TYPE M2MultiplexerProcesses :
STRUCT
	///Select an axis
	selectAxis: M2SelectAxisProcess;
END_STRUCT
END_TYPE

(* stored: Version 1.1.0.1, ProductVersion 3.1.4019.2
   DUT M2MultiplexerProcesses: Id {a64b9fa3-a29d-4f3e-a27a-d6892142ac08} *)
